ABB RAPID module: Module1.mod

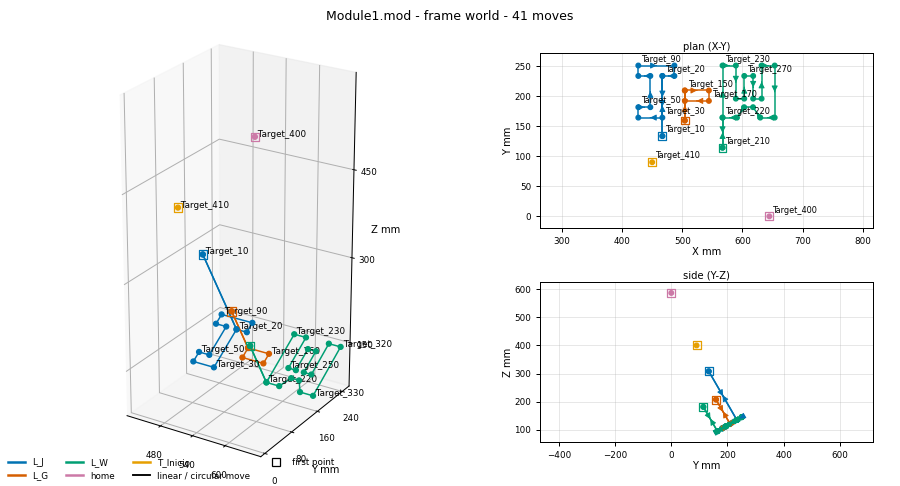
[picture p0: tool path of Module1.mod in frame world, 41 of 41 moves have a stored position in this frame; points joined in program order, loops and branches not executed]
MODULE Module1
        CONST robtarget Target_10:=[[74.615810519,79.997268516,200.000250333],[0.000000516,-0.070288075,0.997526735,-0.000000036],[0,0,0,0],[9E+09,9E+09,9E+09,9E+09,9E+09,9E+09]];
    CONST robtarget Target_20:=[[74.616017354,79.997268516,0.000250333],[0.000000516,-0.070288075,0.997526735,-0.000000036],[0,0,0,0],[9E+09,9E+09,9E+09,9E+09,9E+09,9E+09]];
    CONST robtarget Target_30:=[[154.616017355,79.997268516,0.000333067],[0.000000516,-0.070288075,0.997526735,-0.000000036],[0,0,0,0],[9E+09,9E+09,9E+09,9E+09,9E+09,9E+09]];
    CONST robtarget Target_40:=[[154.616017355,39.997268516,0.000333067],[0.000000516,-0.070288075,0.997526735,-0.000000036],[0,0,0,0],[9E+09,9E+09,9E+09,9E+09,9E+09,9E+09]];
    CONST robtarget Target_50:=[[134.616017354,39.997268516,0.000312384],[0.000000516,-0.070288075,0.997526735,-0.000000036],[0,0,0,0],[9E+09,9E+09,9E+09,9E+09,9E+09,9E+09]];
    CONST robtarget Target_60:=[[134.616017354,59.997268516,0.000312384],[0.000000516,-0.070288075,0.997526735,-0.000000036],[0,0,0,0],[9E+09,9E+09,9E+09,9E+09,9E+09,9E+09]];
    CONST robtarget Target_70:=[[74.616017354,59.997268516,0.000250333],[0.000000516,-0.070288075,0.997526735,-0.000000036],[0,0,0,0],[9E+09,9E+09,9E+09,9E+09,9E+09,9E+09]];
    CONST robtarget Target_80:=[[74.616017354,39.997268516,0.000250333],[0.000000516,-0.070288075,0.997526735,-0.000000036],[0,0,0,0],[9E+09,9E+09,9E+09,9E+09,9E+09,9E+09]];
    CONST robtarget Target_90:=[[54.616017355,39.997268516,0.00022965],[0.000000516,-0.070288075,0.997526735,-0.000000036],[0,0,0,0],[9E+09,9E+09,9E+09,9E+09,9E+09,9E+09]];
    CONST robtarget Target_100:=[[54.616017355,99.997268516,0.00022965],[0.000000516,-0.070288075,0.997526735,-0.000000036],[0,0,0,0],[9E+09,9E+09,9E+09,9E+09,9E+09,9E+09]];
    CONST robtarget Target_110:=[[74.616017354,99.997268516,0.000250333],[0.000000516,-0.070288075,0.997526735,-0.000000036],[0,0,0,0],[9E+09,9E+09,9E+09,9E+09,9E+09,9E+09]];
    CONST robtarget Target_120:=[[74.616017354,79.997268516,0.000250333],[0.000000516,-0.070288075,0.997526735,-0.000000036],[0,0,0,0],[9E+09,9E+09,9E+09,9E+09,9E+09,9E+09]];
    CONST robtarget Target_130:=[[74.615810519,79.997268516,200.000250333],[0.000000516,-0.070288075,0.997526735,-0.000000036],[0,0,0,0],[9E+09,9E+09,9E+09,9E+09,9E+09,9E+09]];
    CONST robtarget Target_140:=[[102.522239363,117.335217332,100.000279194],[0.000000516,-0.070288029,0.997526738,-0.000000036],[0,0,0,0],[9E+09,9E+09,9E+09,9E+09,9E+09,9E+09]];
    CONST robtarget Target_150:=[[102.52234278,117.335217332,0.000279194],[0.000000516,-0.070288029,0.997526738,-0.000000036],[0,0,0,0],[9E+09,9E+09,9E+09,9E+09,9E+09,9E+09]];
    CONST robtarget Target_160:=[[102.52234278,157.335217332,0.000279194],[0.000000516,-0.070288029,0.997526738,-0.000000036],[0,0,0,0],[9E+09,9E+09,9E+09,9E+09,9E+09,9E+09]];
    CONST robtarget Target_170:=[[122.522342779,157.335217332,0.000299877],[0.000000516,-0.070288029,0.997526738,-0.000000036],[0,0,0,0],[9E+09,9E+09,9E+09,9E+09,9E+09,9E+09]];
    CONST robtarget Target_180:=[[122.522342779,117.335217332,0.000299877],[0.000000516,-0.070288029,0.997526738,-0.000000036],[0,0,0,0],[9E+09,9E+09,9E+09,9E+09,9E+09,9E+09]];
    CONST robtarget Target_190:=[[102.52234278,117.335217332,0.000279194],[0.000000516,-0.070288029,0.997526738,-0.000000036],[0,0,0,0],[9E+09,9E+09,9E+09,9E+09,9E+09,9E+09]];
    CONST robtarget Target_200:=[[102.522239363,117.335217332,100.000279194],[0.000000516,-0.070288029,0.997526738,-0.000000036],[0,0,0,0],[9E+09,9E+09,9E+09,9E+09,9E+09,9E+09]];
    CONST robtarget Target_210:=[[154.615913937,180.032099392,100.000333067],[0.000000516,-0.070288031,0.997526738,-0.000000036],[0,0,0,0],[9E+09,9E+09,9E+09,9E+09,9E+09,9E+09]];
    CONST robtarget Target_220:=[[154.616017355,180.032099392,0.000333067],[0.000000516,-0.070288031,0.997526738,-0.000000036],[0,0,0,0],[9E+09,9E+09,9E+09,9E+09,9E+09,9E+09]];
    CONST robtarget Target_230:=[[54.616017355,180.032099392,0.00022965],[0.000000516,-0.070288031,0.997526738,-0.000000036],[0,0,0,0],[9E+09,9E+09,9E+09,9E+09,9E+09,9E+09]];
    CONST robtarget Target_240:=[[54.616017355,202.180714048,0.00022965],[0.000000516,-0.070288031,0.997526738,-0.000000036],[0,0,0,0],[9E+09,9E+09,9E+09,9E+09,9E+09,9E+09]];
    CONST robtarget Target_250:=[[118.192724529,202.180714048,0.0002954],[0.000000516,-0.070288031,0.997526738,-0.000000036],[0,0,0,0],[9E+09,9E+09,9E+09,9E+09,9E+09,9E+09]];
    CONST robtarget Target_260:=[[118.192724529,216.180714048,0.0002954],[0.000000516,-0.070288031,0.997526738,-0.000000036],[0,0,0,0],[9E+09,9E+09,9E+09,9E+09,9E+09,9E+09]];
    CONST robtarget Target_270:=[[74.616017354,216.180714048,0.000250333],[0.000000516,-0.070288031,0.997526738,-0.000000036],[0,0,0,0],[9E+09,9E+09,9E+09,9E+09,9E+09,9E+09]];
    CONST robtarget Target_280:=[[74.616017354,230.965722015,0.000250333],[0.000000516,-0.070288031,0.997526738,-0.000000036],[0,0,0,0],[9E+09,9E+09,9E+09,9E+09,9E+09,9E+09]];
    CONST robtarget Target_290:=[[118.192724529,230.965722015,0.0002954],[0.000000516,-0.070288031,0.997526738,-0.000000036],[0,0,0,0],[9E+09,9E+09,9E+09,9E+09,9E+09,9E+09]];
    CONST robtarget Target_300:=[[118.192724529,244.965722015,0.0002954],[0.000000516,-0.070288031,0.997526738,-0.000000036],[0,0,0,0],[9E+09,9E+09,9E+09,9E+09,9E+09,9E+09]];
    CONST robtarget Target_310:=[[54.616017355,244.965722015,0.00022965],[0.000000516,-0.070288031,0.997526738,-0.000000036],[0,0,0,0],[9E+09,9E+09,9E+09,9E+09,9E+09,9E+09]];
    CONST robtarget Target_320:=[[54.616017355,266.75931277,0.00022965],[0.000000516,-0.070288031,0.997526738,-0.000000036],[0,0,0,0],[9E+09,9E+09,9E+09,9E+09,9E+09,9E+09]];
    CONST robtarget Target_330:=[[154.616017355,266.75931277,0.000333067],[0.000000516,-0.070288031,0.997526738,-0.000000036],[0,0,0,0],[9E+09,9E+09,9E+09,9E+09,9E+09,9E+09]];
    CONST robtarget Target_340:=[[154.616017355,242.75931277,0.000333067],[0.000000516,-0.070288031,0.997526738,-0.000000036],[0,0,0,0],[9E+09,9E+09,9E+09,9E+09,9E+09,9E+09]];
    CONST robtarget Target_350:=[[134.616017354,230.75931277,0.000312384],[0.000000515,-0.070288031,0.997526738,-0.000000036],[0,0,0,0],[9E+09,9E+09,9E+09,9E+09,9E+09,9E+09]];
    CONST robtarget Target_360:=[[134.616017354,216.032099392,0.000312384],[0.000000516,-0.070288031,0.997526738,-0.000000036],[0,0,0,0],[9E+09,9E+09,9E+09,9E+09,9E+09,9E+09]];
    CONST robtarget Target_370:=[[154.616017355,204.032099392,0.000333067],[0.000000423,-0.070288031,0.997526738,-0.000000296],[0,0,0,0],[9E+09,9E+09,9E+09,9E+09,9E+09,9E+09]];
    CONST robtarget Target_380:=[[154.616017355,180.032099392,0.000333067],[0.000000516,-0.070288031,0.997526738,-0.000000036],[0,0,0,0],[9E+09,9E+09,9E+09,9E+09,9E+09,9E+09]];
    CONST robtarget Target_390:=[[154.615913937,180.032099392,100.000333067],[0.000000516,-0.070288031,0.997526738,-0.000000036],[0,0,0,0],[9E+09,9E+09,9E+09,9E+09,9E+09,9E+09]];
    CONST robtarget Target_400:=[[50.707217621,257.933675895,508.375664587],[0.270598388,-0.701057337,0.653281342,-0.092296318],[0,0,0,0],[9E+09,9E+09,9E+09,9E+09,9E+09,9E+09]];
    CONST robtarget Target_410:=[[66.220306768,63.072,301.506592597],[0.401971692,0.638986864,-0.581737706,-0.302813124],[0,0,0,0],[9E+09,9E+09,9E+09,9E+09,9E+09,9E+09]];
!***********************************************************
    !
    ! Módulo:  Module1
    !
    ! Descripción:
    !   <Introduzca la descripción aquí>
    !
    ! Autor: javie
    !
    ! Versión: 1.0
    !
    !***********************************************************


    !***********************************************************
    !
    ! Procedimiento Main
    !
    !   Este es el punto de entrada de su programa
    !
    !***********************************************************
    PROC main()
        !Añada aquí su código
        home;
        T_Inicio;
        L_J;
        L_G;
        L_W;
        T_Inicio;
        home;
    ENDPROC
    PROC L_J()
        MoveL Target_10,v100,z10,TCP_M\WObj:=WO_M;
        MoveL Target_20,v100,z10,TCP_M\WObj:=WO_M;
        MoveL Target_30,v100,z10,TCP_M\WObj:=WO_M;
        MoveL Target_40,v100,z10,TCP_M\WObj:=WO_M;
        MoveL Target_50,v100,z10,TCP_M\WObj:=WO_M;
        MoveL Target_60,v100,z10,TCP_M\WObj:=WO_M;
        MoveL Target_70,v100,z10,TCP_M\WObj:=WO_M;
        MoveL Target_80,v100,z10,TCP_M\WObj:=WO_M;
        MoveL Target_90,v100,z10,TCP_M\WObj:=WO_M;
        MoveL Target_100,v100,z10,TCP_M\WObj:=WO_M;
        MoveL Target_110,v100,z10,TCP_M\WObj:=WO_M;
        MoveL Target_120,v100,z10,TCP_M\WObj:=WO_M;
        MoveL Target_130,v100,z10,TCP_M\WObj:=WO_M;
    ENDPROC
    PROC L_G()
        MoveL Target_140,v100,z10,TCP_M\WObj:=WO_M;
        MoveL Target_150,v100,z10,TCP_M\WObj:=WO_M;
        MoveL Target_160,v100,z10,TCP_M\WObj:=WO_M;
        MoveL Target_170,v100,z10,TCP_M\WObj:=WO_M;
        MoveL Target_180,v100,z10,TCP_M\WObj:=WO_M;
        MoveL Target_190,v100,z10,TCP_M\WObj:=WO_M;
        MoveL Target_200,v100,z10,TCP_M\WObj:=WO_M;
    ENDPROC
    PROC L_W()
        MoveL Target_210,v100,z10,TCP_M\WObj:=WO_M;
        MoveL Target_220,v100,z10,TCP_M\WObj:=WO_M;
        MoveL Target_230,v100,z10,TCP_M\WObj:=WO_M;
        MoveL Target_240,v100,z10,TCP_M\WObj:=WO_M;
        MoveL Target_250,v100,z10,TCP_M\WObj:=WO_M;
        MoveL Target_260,v100,z10,TCP_M\WObj:=WO_M;
        MoveL Target_270,v100,z10,TCP_M\WObj:=WO_M;
        MoveL Target_280,v100,z10,TCP_M\WObj:=WO_M;
        MoveL Target_290,v100,z10,TCP_M\WObj:=WO_M;
        MoveL Target_300,v100,z10,TCP_M\WObj:=WO_M;
        MoveL Target_310,v100,z10,TCP_M\WObj:=WO_M;
        MoveL Target_320,v100,z10,TCP_M\WObj:=WO_M;
        MoveL Target_330,v100,z10,TCP_M\WObj:=WO_M;
        MoveL Target_340,v100,z10,TCP_M\WObj:=WO_M;
        MoveL Target_350,v100,z10,TCP_M\WObj:=WO_M;
        MoveL Target_360,v100,z10,TCP_M\WObj:=WO_M;
        MoveL Target_370,v100,z10,TCP_M\WObj:=WO_M;
        MoveL Target_380,v100,z10,TCP_M\WObj:=WO_M;
        MoveL Target_390,v100,z10,TCP_M\WObj:=WO_M;
    ENDPROC
    PROC home()
        MoveL Target_400,v1000,z100,TCP_M\WObj:=WO_M;
    ENDPROC
    PROC T_Inicio()
        MoveL Target_410,v1000,z100,TCP_M\WObj:=WO_M;
    ENDPROC
ENDMODULE
